{attribute 'qualified_only'}
{attribute 'strict'}
TYPE eWago750495_StatDataID_1 :
(
	Phase1 := 0,
	Phase2 := 1,
	Phase3 := 2,
	IOmodule:= 3
)USINT;
END_TYPE

(* stored: Version 1.1.0.1, ProductVersion 3.1.4024.12
   DUT eWago750495_StatDataID_1: Id {712203a5-c89f-40e3-a646-591a2f468333} *)
